TYPE Bits8 :
STRUCT
	Bit0 : BIT;
	Bit1 : BIT;
	Bit2 : BIT;
	Bit3 : BIT;
	Bit4 : BIT;
	Bit5 : BIT;
	Bit6 : BIT;
	Bit7 : BIT;
END_STRUCT
END_TYPE

(* stored: Version 1.1.0.1
   DUT Bits8: Id {e42a0440-51a1-0790-010f-36417b434ebd} *)
